# B&R Automation Studio project Test_V6x
Automation Studio 6.5.0.306; technology packages: mappMotion 6.5.1, mappSafety 6.4.1, OpcUaCs 6.4.0

## Configuration Config1

CPU PC_any, AutomationRuntime 6.4.2, Build 11.3.0, Vc 6.0.0

### Task classes (AppMo.sw)
```
Cyclic#1:
  myApptask1 <- myAppMod1.myApptask1.prg
```

### Task classes (Cpu.sw)
```
Cyclic#1:
  Axes <- MotionHandling.Axes.prg
DataObjects: McAcpSys
NcDataObjects: McDriveLog
Binaries: udbdef, ArSvcReg, FWRules, McProfGen, McAcpSim, McAcpDrv, TCData, iomap, asfw, ashwd, UaCsConfig, BRRole, Config_1, arconfig, ashwac, sysconf
Libraries: SfDomain, MpBase, McBase, MpAxis, McAxis, McAcpAx, McAxGroup, McPureVAx, UaCoal, UaCore, standard, SfDomVis, MpSfDomMgr, fileio, powerlnk, AsIODiag, AsIOAcc, SfDomDrv, sys_lib, ArUser, astime, UaCoalPrv, runtime, AsEPL, AsUSB, AsTCP
```

### Hardware
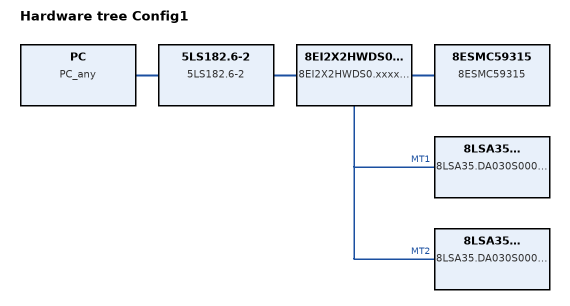
```
5LS182.6-2 : 5LS182.6-2 v1.13.0.0  [SL -> PC.SL1]
8EI2X2HWDS0.xxxx-1 : 8EI2X2HWDS0.xxxx-1 v2.5.0.0 (NodeNumber=1)  [PLK1 -> 5LS182.6-2.IF1 [Cable Type=PowerlinkCable, Length=10, Version=1.0.0.3]; MT2 -> 8LSA35.DA030S000-3_a.MT]
8ESMC59315 : 8ESMC59315 v2.6.0.0  [SafeMOTION -> 8EI2X2HWDS0.xxxx-1.SafeMOTION1]
8LSA35.DA030S000-3 : 8LSA35.DA030S000-3 v2.2.0.2  [MT -> 8EI2X2HWDS0.xxxx-1.MT1]
  M1/MotorParameters:
    MOTOR_AMB_TEMP_RATED = 40
  M1/MotorParameters/TemperatureSensor:
    MOTOR_TEMPSENS_LIM = 130
8LSA35.DA030S000-3_a : 8LSA35.DA030S000-3 v2.2.0.2  [MT -> 8EI2X2HWDS0.xxxx-1.MT2]
  M1/MotorParameters:
    MOTOR_AMB_TEMP_RATED = 40
  M1/MotorParameters/TemperatureSensor:
    MOTOR_TEMPSENS_LIM = 130
PC : PC_any v1.1.2.0 (OrderNumber=PC)
  ConfigurationID = test_Config1
  VolatileGlobalPvSize = 256000
  FileDevice1
  FileDeviceName1 = USER
  FileDevicePath1 = USER_PATH
```

### BRRole.brrole - PC/AccessAndSecurity/UserRoleSystem/BRRole.brrole
```
Element BR_Anonymous (Type=BRRole)
Element BR_Engineer (Type=BRRole)
Element BR_Observer (Type=BRRole)
Element BR_SafetyAdmin (Type=BRRole)
Element BR_SecurityAdmin (Type=BRRole)
```

### Config_1.axis - PC/mappMotion/Config_1.axis
```
Element gAxisY (Type=axis)
Element gAxisX (Type=axis)
```

## Logical view

Binary libraries used (declarations not repeated): operator, runtime, AsIecCon, astime, SfDomain 6.4.1, MpBase 6.5.0, McBase 6.5.1, MpAxis 6.5.1, McAxis 6.5.1, McAcpAx 6.5.1, McAxGroup 6.5.1, McPureVAx 6.5.1

### Package Logical/Libraries - Global libraries

### MotionHandling.typ
```iecst
TYPE
	AxisHandlingAxesGroupStepEnum :
		(
		AHG_W_EVENT, (*warte auf Ereignis*)
		AHG_READ_NEXT_ERROR_RECORD, (*nächsten Fehlerdatensatz lesen*)
		AHG_COPY_ERROR_RECORDS, (*kopiere alle Fehlerinformationen*)
		AHG_W_RESET (*alle Fehlertexte wurden gelesen*)
		);
	AxisHandlingAxesStepEnum :
		(
		AX_STARTUP,
		AX_W_CONFIGURATION_READ,
		AX_W_EVENT, (*warte auf Ereignis*)
		AX_READ_NEXT_ERROR_RECORD, (*nächsten Fehlerdatensatz lesen*)
		AX_COPY_ERROR_RECORDS, (*kopiere alle Fehlerinformationen*)
		AX_W_RESET, (*alle Fehlertexte wurden gelesen*)
		AX_WRITE_CONFIGURATION (*schreibe neue Achskonfiguration*)
		);
	AxisHandlingAxisType : 	STRUCT
		name : STRING[32];
		step : AxisHandlingAxesStepEnum; (*Schrittkette*)
		errorTextHeader : STRING[80];
		errorText : STRING[16384]; (*Fehlertexte*)
		errorTextLines : UINT; (*Fehlertexte: Anzahl der Zeilen*)
		pAxis : UDINT;
		fbMpAxis : MpAxisBasic;
		mpAxisParameters : MpAxisBasicParType;
		fbMoveAbsolute : MC_MoveAbsolute;
		nullpos : LREAL; (*Fahrt auf diese Position nach Homing*)
		pureVaxAdapter : McPureVAxDS402VlAdapterPvType;
		statusInputSTO : BOOL; (*Status STO/Enable*)
		fbForceHardwareInputs : MC_BR_ForceHardwareInputs;
		fbMpAxisBasicConfig : MpAxisBasicConfig;
		mpAxisBasicConfigData : MpAxisBasicConfigType;
		fbReadErrorText : MC_BR_ReadErrorText;
		fbCommandError : MC_BR_CommandError;
		n : UINT;
	END_STRUCT;
	AxisHandlingAxesGroupType : 	STRUCT
		name : STRING[32];
		step : AxisHandlingAxesGroupStepEnum; (*Schrittkette*)
		errorTextHeader : STRING[80];
		errorText : STRING[16384]; (*Fehlertexte*)
		errorTextLines : UINT; (*Fehlertexte: Anzahl der Zeilen*)
		pAxGroup : UDINT;
		fbGroupPower : MC_BR_GroupPower;
		fbGroupHome : MC_BR_GroupHome_15;
		fbGroupReset : MC_GroupReset;
		fbGroupReadInfo : MC_BR_GroupReadInfo;
		fbGroupReadStatus : MC_GroupReadStatus;
		fbReadErrorText : MC_BR_ReadErrorText;
		n : UINT;
	END_STRUCT;
	AxisHandlingType : 	STRUCT
		ax : ARRAY[0..MAX_AX_MINUS_ONE]OF AxisHandlingAxisType;
		axGroupCnc : AxisHandlingAxesGroupType;
		axGroupAux : AxisHandlingAxesGroupType;
	END_STRUCT;
END_TYPE
```

### MotionHandling.var
```iecst
VAR CONSTANT
	MAX_AX : USINT := 2;
	MAX_AX_MINUS_ONE : USINT := MAX_AX-1;
END_VAR
VAR
	gAxisHandling : AxisHandlingType;
END_VAR
VAR CONSTANT
	AX_X : USINT := 0;
	AX_Y : USINT := 1;
END_VAR
```

### Program Logical/MotionHandling/Axes (IEC) - Achsen und Achsengruppen

#### Variables.var
```iecst
VAR
	ax : REFERENCE TO AxisHandlingAxisType;
	axX : REFERENCE TO AxisHandlingAxisType; (*OPCUa tag*)
	axY : REFERENCE TO AxisHandlingAxisType; (*OPCUa tag*)
	size1 : UDINT;
END_VAR
```

#### Main.st
```iecst
PROGRAM _INIT
	gAxisHandling.ax[AX_X].name := 'X';
	gAxisHandling.ax[AX_X].pAxis := ADR(gAxisX);
	axX ACCESS ADR(gAxisHandling.ax[AX_X]);

	size1 := SIZEOF(axX);
	axX.n := 99;

	gAxisHandling.ax[AX_Y].name := 'Y';
	gAxisHandling.ax[AX_Y].pAxis := ADR(gAxisY);
	axY ACCESS ADR(gAxisHandling.ax[AX_Y]);

END_PROGRAM

PROGRAM _CYCLIC

END_PROGRAM

PROGRAM _EXIT

END_PROGRAM
```

### Program Logical/myAppMod1/myApptask1 (IEC)

#### Variables.var
```iecst
VAR
	i : USINT := 0;
END_VAR
```

#### Main.st
```iecst
PROGRAM _INIT
	(* Insert code here *)

END_PROGRAM

PROGRAM _CYCLIC
	i := i + 1;

END_PROGRAM

PROGRAM _EXIT
	(* Insert code here *)

END_PROGRAM
```

### Program Logical/Programs/myProg (IEC) - Program

#### Type.typ - Local data types
```iecst
TYPE
	myStructType : 	STRUCT
		member1 : USINT := 3;
		member2 : ARRAY[0..2]OF USINT := [33,44,55];
	END_STRUCT;
	myEnumType :
		(
		eins,
		zwei,
		drei
		);
	myDerivedType1 :USINT(4..6) ;
	myDerivedType :ARRAY[3..6]OF USINT;
	myComplexStructType : 	STRUCT
		element : USINT;
		vector : ARRAY[1..10]OF REAL;
		matrix : ARRAY[0..9,0..3]OF REAL;
		myStruct0 : myStructType;
		myStruct1 : ARRAY[0..1]OF myStructType;
		myStruct2 : ARRAY[2..2]OF myStructType;
		myStruct3 : ARRAY[-1..1]OF myStructType;
		myStruct4 : ARRAY[0..2,0..3]OF myStructType;
		myEnum : myEnumType;
		subrange1 : SINT(-3..6) ;
		derived1 : myDerivedType1;
		myDerived1 : myDerivedType;
		n : USINT := 99;
	END_STRUCT;
END_TYPE
```

#### myProg.st - Implementation code
```iecst
(********************************************************************
 * COPYRIGHT -- B&R Industrial Automation GmbH
 ********************************************************************
 * Program: myProg
 * File: myProg.st
 * Author: hilchenbachc
 * Created: November 22, 2022
 ********************************************************************
 * Implementation of program myProg
 ********************************************************************)

PROGRAM _INIT
	myUSINT := 91;
	myUINT := 92;
	mySTRING := 'Hello, world';
	myWSTRING := "Hello, world";
	myTIME := T#314s;
	myTOD := TOD#14:15:30.000;
	myDT := DT#2025-02-07-06:28:15;
	myDINT := -93;
	myINTArray;
	mySTRINGArray;
	myWSTRINGArray;
	myUDINT := 94;
	myDATE := D#2025-02-07 ;
	myLREAL := 95.6;
	myREAL := 96.7;
	myINT := 97;
	mySINT := 98;
	myBOOL := TRUE;
	myStructArray;

	FOR i := 0 TO 9 DO
		myComplexStruct.vector[i+1] := 200 + i;
		FOR j := 0 TO 3 DO
			myComplexStruct.matrix[i,j] := 1000 + (10 * i + j);
		END_FOR
	END_FOR
	myComplexStruct.myEnum := drei;
	sizeof_myComplexStruct := SIZEOF(myComplexStruct);

END_PROGRAM

PROGRAM _CYCLIC

END_PROGRAM
```

#### myProg.var - Local variables
```iecst
(********************************************************************
 * COPYRIGHT -- B&R Industrial Automation GmbH
 ********************************************************************
 * Program: myProg
 * File: myProg.var
 * Author: hilchenbachc
 * Created: November 22, 2022
 ********************************************************************
 * Local variables of program myProg
 ********************************************************************)
VAR
	myUSINT : USINT := 0;
	myUINT : UINT := 0;
	mySTRING : STRING[80] := '';
	myWSTRING : WSTRING[80] := "";
	myTIME : TIME := T#0S;
	myTOD : TIME_OF_DAY := TOD#00:00:00;
	myDT : DATE_AND_TIME := DT#1970-01-01-00:00:00;
	myDINT : DINT := 0;
	myINTArray : ARRAY[0..9] OF INT := [10(0)];
	myWSTRINGArray : ARRAY[0..9] OF WSTRING[80];
	mySTRINGArray : ARRAY[0..9] OF STRING[80];
	myUDINT : UDINT := 0;
	myDATE : DATE;
	myLREAL : LREAL := 0.0;
	myREAL : REAL := 0.0;
	myINT : INT := 0;
	mySINT : SINT := 0;
	myBOOL : BOOL := FALSE;
	myStructArray : ARRAY[0..1] OF myStructType;
	myComplexStruct : myComplexStructType;
	i : INT;
	j : INT;
	sizeof_myComplexStruct : UDINT;
END_VAR
```

Listed in the project but not available here: Logical/Global.var
